{attribute addProperty BoxType "EK1100-0000-0018"}
{attribute addProperty Id "Beckhoff_EJx9xxEK1122Beckhoff_EJx9xxEK1122_05D2B413162A_0001_EJ1914_0000_0017EJ1914_8416AE0F22428A_0002_EJ1914_0000_0018EJ1914_8416AE0F22428A_0003_EJ1918_0000_0017EJ1918_6B01E91023229A_0004_EJ1918_0000_0018EJ1918_6B01E91023229A_0005_EJ1957_0000_0017EJ1957_FBD97F1D28836A_0006_EJ1957_0000_0018EJ1957_FBD97F1D28836A_0007_EJ2914_0000_0017EJ2914_26D491F127234A_0008_EJ2914_0000_0018EJ2914_26D491F127234A_0009_EJ2918_0000_0017EJ2918_C5F09C7031239A_0010_EJ2918_0000_0018EJ2918_C5F09C7031239A_0011_EJ6910_0000_0018EJ6910_13AA933411214A_0012_EJ6910_0000_0020EJ6910_13AA933411214"}
{attribute addProperty CRC "1741030744"}
{attribute addProperty SizeInBites "2896"}
{attribute addProperty SizeInBytes "362"}
TYPE Beckhoff_EJx9xx_67C60558 EXTENDS EK1100_179A0949 :
STRUCT
	{attribute addProperty Name "Beckhoff_EJx9xxEK1122"}
	Beckhoff_EJx9xxEK1122 : Beckhoff_EJx9xxEK1122_05D2B413;
	{attribute addProperty Name "A_0001_EJ1914_0000_0017"}
	A_0001_EJ1914_0000_0017 : EJ1914_8416AE0F;
	{attribute addProperty Name "A_0002_EJ1914_0000_0018"}
	A_0002_EJ1914_0000_0018 : EJ1914_8416AE0F;
	{attribute addProperty Name "A_0003_EJ1918_0000_0017"}
	A_0003_EJ1918_0000_0017 : EJ1918_6B01E910;
	{attribute addProperty Name "A_0004_EJ1918_0000_0018"}
	A_0004_EJ1918_0000_0018 : EJ1918_6B01E910;
	{attribute addProperty Name "A_0005_EJ1957_0000_0017"}
	A_0005_EJ1957_0000_0017 : EJ1957_FBD97F1D;
	{attribute addProperty Name "A_0006_EJ1957_0000_0018"}
	A_0006_EJ1957_0000_0018 : EJ1957_FBD97F1D;
	{attribute addProperty Name "A_0007_EJ2914_0000_0017"}
	A_0007_EJ2914_0000_0017 : EJ2914_26D491F1;
	{attribute addProperty Name "A_0008_EJ2914_0000_0018"}
	A_0008_EJ2914_0000_0018 : EJ2914_26D491F1;
	{attribute addProperty Name "A_0009_EJ2918_0000_0017"}
	A_0009_EJ2918_0000_0017 : EJ2918_C5F09C70;
	{attribute addProperty Name "A_0010_EJ2918_0000_0018"}
	A_0010_EJ2918_0000_0018 : EJ2918_C5F09C70;
	{attribute addProperty Name "A_0011_EJ6910_0000_0018"}
	A_0011_EJ6910_0000_0018 : EJ6910_13AA9334;
	{attribute addProperty Name "A_0012_EJ6910_0000_0020"}
	A_0012_EJ6910_0000_0020 : EJ6910_13AA9334;
END_STRUCT
END_TYPE

(* stored: Version 1.2.0.0, ProductVersion 3.1.4024.9
   DUT Beckhoff_EJx9xx_67C60558: Id {437b3755-11c6-456c-b9f4-bc58b25be534} *)
